Staubli VAL3: Form_6jHome.pgx

public program Form_6jHome(string x_sTitle, jointRx& x_jJ)
begin

  call Form_PattenS(x_sTitle,"记录,,,,,上传,保存,退出","记录,,,,,上传,保存,退出")
  call Control_PanelXY(22,0,15,10)
  call Control_Panel("Home")
  //call con
  gotoxy(nPanelLTopX+1,nPanelLTopY+1)
  put(left("j1:"+toString(".3",x_jJ.j1)+"        ",nPanelWidthX))

  gotoxy(nPanelLTopX+1,nPanelLTopY+2)
  put(left("j2:"+toString(".3",x_jJ.j2)+"        ",nPanelWidthX))

  gotoxy(nPanelLTopX+1,nPanelLTopY+3)
  put(left("j3:"+toString(".3",x_jJ.j3)+"        ",nPanelWidthX))

  gotoxy(nPanelLTopX+1,nPanelLTopY+4)
  put(left("j4:"+toString(".3",x_jJ.j4)+"        ",nPanelWidthX))


  gotoxy(nPanelLTopX+1,nPanelLTopY+5)
  put(left("j5:"+toString(".3",x_jJ.j5)+"        ",nPanelWidthX))

  gotoxy(nPanelLTopX+1,nPanelLTopY+6)
  put(left("j6:"+toString(".3",x_jJ.j6)+"        ",nPanelWidthX))



end
